FUNCTION_BLOCK TEST_MOD (* Test modulo functions *)
  (* Standard: 61499-2 *)
  (* Version 0.0, 2006-09-05, JHC, Holobloc Inc *)
  (* Compiler header: package fb.rt.test; *)
  (* Compiler classdef: public class TEST_ABS extends SimpleFB *)
  (* Compiler Java Sun JDK 1.5.0 *)
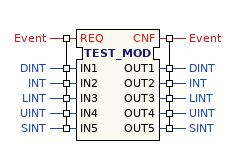
  EVENT_INPUT
    REQ WITH IN1, IN2, IN3, IN4, IN5; (* Normal Execution Request *)
  END_EVENT
  EVENT_OUTPUT
    CNF WITH OUT1, OUT2, OUT3, OUT4, OUT5; (* Execution Confirmation *)
  END_EVENT
  VAR_INPUT
    IN1 : DINT;
    IN2 : INT;
    IN3 : LINT;
    IN4 : UINT;
    IN5 : SINT;
  END_VAR
  VAR_OUTPUT
    OUT1 : DINT;
    OUT2 : INT;
    OUT3 : LINT;
    OUT4 : UINT;
    OUT5 : SINT;
  END_VAR
  ALGORITHM REQ IN FBD: (* Normally executed algorithm *)
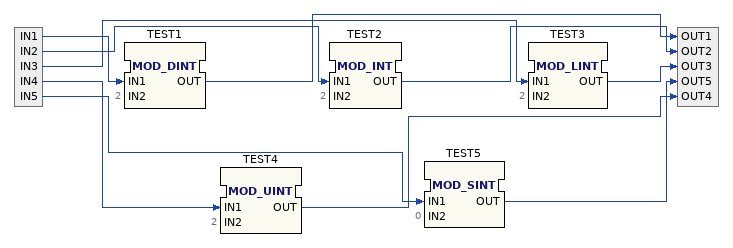
    FBS
      TEST1 : MOD_DINT(IN2 := 2);
      TEST2 : MOD_INT(IN2 := 2);
      TEST3 : MOD_LINT(IN2 := 2);
      TEST4 : MOD_UINT(IN2 := 2);
      TEST5 : MOD_SINT(IN2 := 0);
    END_FBS
    DATA_CONNECTIONS
      TEST1.OUT TO OUT1;
      TEST2.OUT TO OUT2;
      TEST3.OUT TO OUT3;
      TEST5.OUT TO OUT5;
      IN1 TO TEST1.IN1;
      IN2 TO TEST2.IN1;
      IN3 TO TEST3.IN1;
      IN4 TO TEST4.IN1;
      TEST4.OUT TO OUT4;
      IN5 TO TEST5.IN1;
    END_CONNECTIONS
  END_ALGORITHM
END_FUNCTION_BLOCK
